Fanuc KAREL source: FORMAT_DEV.kl

PROGRAM T
%NOLOCKGROUP
VAR
 v0 : STRING[40]
 v1 : STRING[40]
 v2 : BOOLEAN
 v3 : INTEGER
BEGIN
 FORMAT_DEV(v0, v1, v2, v3)
END T
